// Mitsubishi GX Works2 project: Lab_3_insys_P_J   PLC: FX1N/FX1NC

// global labels: Global1
VAR_GLOBAL
  stopp AT X000 : BOOL;
  start AT X001 : BOOL;
  motorvern AT X002 : BOOL;
  endebryter_A_tilbake AT X003 : BOOL;
  endebryter_A_fremme AT X004 : BOOL;
  endebryter_Bor_nede AT X005 : BOOL;
  endebryter_Bor_oppe AT X006 : BOOL;
  endebryter_C_tilbake AT X007 : BOOL;
  endebryter_C_fremme AT X010 : BOOL;
  kontaktor_K1 AT Y000 : BOOL;
  A_frem AT Y001 : BOOL;
  A_tilbake AT Y002 : BOOL;
  Bor_opp AT Y003 : BOOL;
  Bor_ned AT Y004 : BOOL;
  C_frem AT Y005 : BOOL;
  C_tilbake AT Y006 : BOOL;
END_VAR

// task Task_01 (event TRUE, interval 0, priority 31): borelabb

PROGRAM borelabb
(* structured ladder/FBD written out as ST: instructions are called as NAME(EN, inputs, outputs); _pN, _eN, _tN stand for wires *)
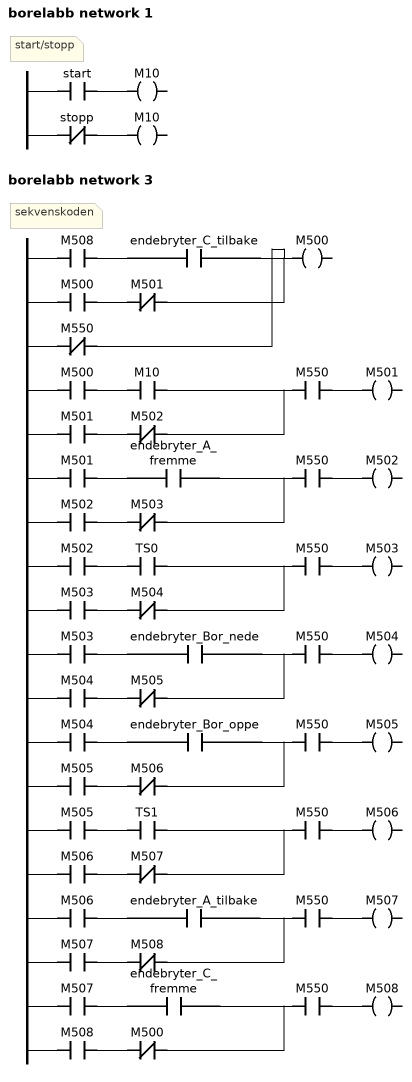
(* network 1 *)
(* start/stopp *)
M10 := start;
M10 := NOT stopp;
(* jump greier *)
(* network 3 *)
(* sekvenskoden *)
M500 := (M508 AND endebryter_C_tilbake) OR (M500 AND NOT M501) OR (NOT M550);
M501 := ((M500 AND M10) OR (M501 AND NOT M502)) AND M550;
M502 := ((M501 AND endebryter_A_fremme) OR (M502 AND NOT M503)) AND M550;
M503 := ((M502 AND TS0) OR (M503 AND NOT M504)) AND M550;
M504 := ((M503 AND endebryter_Bor_nede) OR (M504 AND NOT M505)) AND M550;
M505 := ((M504 AND endebryter_Bor_oppe) OR (M505 AND NOT M506)) AND M550;
M506 := ((M505 AND TS1) OR (M506 AND NOT M507)) AND M550;
M507 := ((M506 AND endebryter_A_tilbake) OR (M507 AND NOT M508)) AND M550;
M508 := ((M507 AND endebryter_C_fremme) OR (M508 AND NOT M500)) AND M550;
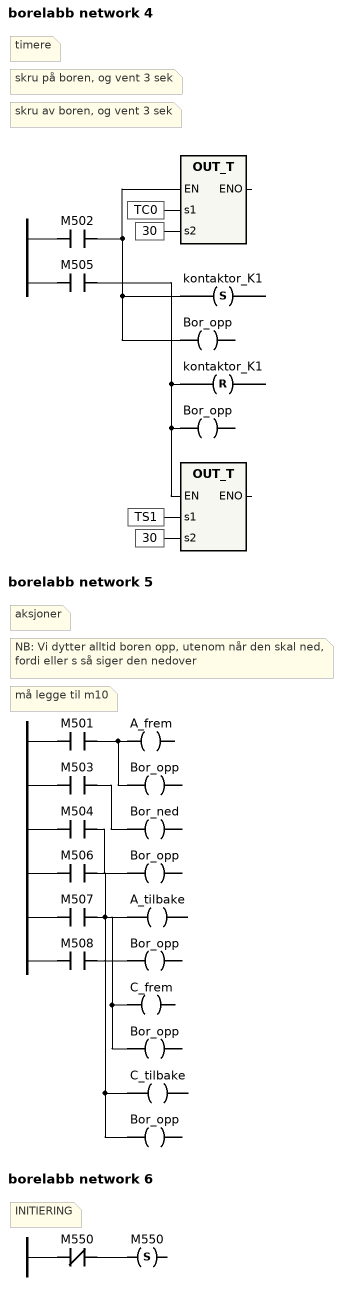
(* network 4 *)
(* timere *)
(* skru på boren, og vent 3 sek *)
(* skru av boren, og vent 3 sek *)
SET(M502, kontaktor_K1);
Bor_opp := M502;
OUT_T(M502, TC0, 30);
RST(M505, kontaktor_K1);
Bor_opp := M505;
OUT_T(M505, TS1, 30);
(* network 5 *)
(* aksjoner *)
(* NB: Vi dytter alltid boren opp, utenom når den skal ned, fordi eller s så siger den nedover *)
(* må legge til m10 *)
A_frem := M501;
Bor_opp := M501;
Bor_ned := M503;
Bor_opp := M504;
A_tilbake := M506;
Bor_opp := M506;
C_frem := M507;
Bor_opp := M507;
C_tilbake := M508;
Bor_opp := M508;
(* network 6 *)
(* INITIERING *)
SET(NOT M550, M550);
END_PROGRAM
